(* Logix 5000 project; controller SFC_Machine_Cycle_Portfolio vendor 1 type 14 code 196 rev 36.11; software revision 36.00 *)

TASK MainTask (continuous, watchdog 500 ms) : MainProgram

MODULES
   Local : vendor 1 type 14 code 196 (5069 0, rev 36.11)
END_MODULES

VAR_GLOBAL   (* controller tags *)
   Cycle_Active : BOOL;
   Cycle_Start_Request : BOOL;
   Fault_Active : BOOL;
   Machine_Ready : BOOL;
   Mode_Auto : BOOL;
   PB_Reset : BOOL;
   PB_Start : BOOL;
   PB_Stop : BOOL;
   Stop_Request : BOOL;
END_VAR

PROGRAM MainProgram   (* main routine MainRoutine *)
VAR
   A_Unclamp : SFC_ACTION := (Status := 16#0020_0000, PauseTimer := 1);
   Action_000 : SFC_ACTION := (Status := 16#0020_0000, PauseTimer := 1);
   Clamp_Cmd : BOOL;
   Clamp_Extended_LS : BOOL;
   Clamp_Retracted_LS : BOOL;
   Clamp_Timeout_Fault : BOOL;
   Drill_At_Depth_LS : BOOL;
   Drill_At_Home_LS : BOOL;
   Drill_Fwd_Cmd : BOOL;
   Drill_Retract : SFC_STEP := (Status := 16#0020_0000, PauseTimer := 1);
   Drill_Rev_Cmd : BOOL;
   DrillFwd_Timeout_Fault : BOOL;
   DrillRev_Timeout_Fault : BOOL;
   Eject_Cmd : BOOL;
   Eject_Extend : SFC_STEP := (Status := 16#0020_0000, PauseTimer := 1);
   Eject_Extended_LS : BOOL;
   Eject_Retracted_LS : BOOL;
   EjectExtend_Timeout_Fault : BOOL;
   EjectRetract_Timeout_Fault : BOOL;
   Machine_State : DINT;   // 0 = idle 10 = Clamp 20 = Drill Foward 30 = Drill Retract 40 = Unclamp 50 = Eject Extended 60 = Eject Retract 70 = Complete
   Sim_Enable : BOOL;
   Step_Clamp_Active : BOOL;
   Step_Complete_Active : BOOL;
   Step_DrillFwd_Active : BOOL;
   Step_DrillRev_Active : BOOL;
   Step_EjectExtend_Active : BOOL;
   Step_EjectRetract_Active : BOOL;
   Step_Idle_Active : BOOL;
   Step_Unclamp_Active : BOOL;
   T_Clamp_Extend : TIMER := (PRE := 1000);
   T_Clamp_Retract : TIMER := (PRE := 1000);
   T_Clamp_Timeout : TIMER := (PRE := 3000);
   T_Drill_Fwd : TIMER := (PRE := 3000);
   T_Drill_Rev : TIMER := (PRE := 1500);
   T_DrillFwd_Timeout : TIMER := (PRE := 4000);
   T_DrillRev_Timeout : TIMER := (PRE := 4000);
   T_Eject_Extend : TIMER := (PRE := 1000);
   T_Eject_Retract : TIMER := (PRE := 1000);
   T_EjectExtend_Timeout : TIMER := (PRE := 3000);
   T_EjectRetract_Timeout : TIMER := (PRE := 3000);
   Tran_000 : BOOL;
   Tran_001 : BOOL;
   Unclamp : SFC_STEP := (Status := 16#0020_0000, PauseTimer := 1);
END_VAR

ROUTINE Faults   (* ladder *)
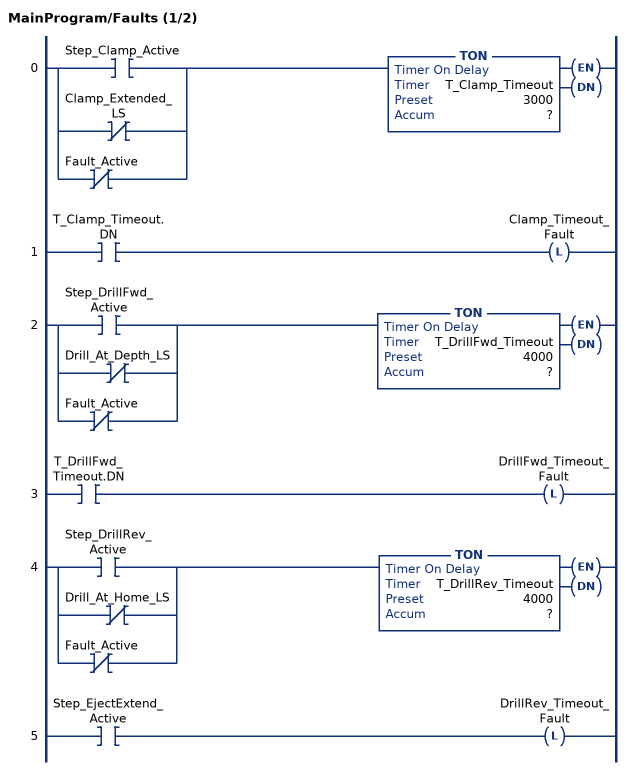
   0: [XIC(Step_Clamp_Active) ,XIO(Clamp_Extended_LS) ,XIO(Fault_Active) ]TON(T_Clamp_Timeout,?,?);
   1: XIC(T_Clamp_Timeout.DN)OTL(Clamp_Timeout_Fault);
   2: [XIC(Step_DrillFwd_Active) ,XIO(Drill_At_Depth_LS) ,XIO(Fault_Active) ]TON(T_DrillFwd_Timeout,?,?);
   3: XIC(T_DrillFwd_Timeout.DN)OTL(DrillFwd_Timeout_Fault);
   4: [XIC(Step_DrillRev_Active) ,XIO(Drill_At_Home_LS) ,XIO(Fault_Active) ]TON(T_DrillRev_Timeout,?,?);
   5: XIC(Step_EjectExtend_Active)OTL(DrillRev_Timeout_Fault);
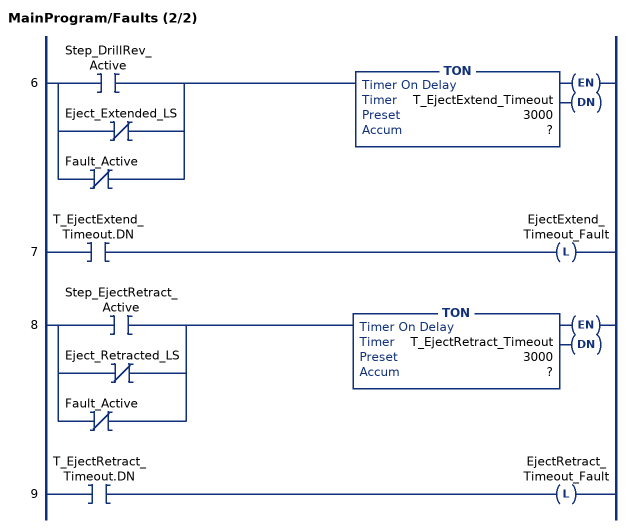
   6: [XIC(Step_DrillRev_Active) ,XIO(Eject_Extended_LS) ,XIO(Fault_Active) ]TON(T_EjectExtend_Timeout,?,?);
   7: XIC(T_EjectExtend_Timeout.DN)OTL(EjectExtend_Timeout_Fault);
   8: [XIC(Step_EjectRetract_Active) ,XIO(Eject_Retracted_LS) ,XIO(Fault_Active) ]TON(T_EjectRetract_Timeout,?,?);
   9: XIC(T_EjectRetract_Timeout.DN)OTL(EjectRetract_Timeout_Fault);
END_ROUTINE

ROUTINE Machine_SFC   (* sequential function chart *)
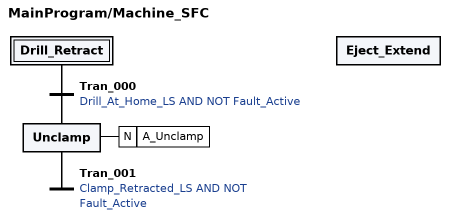
   INITIAL_STEP Drill_Retract:
   END_STEP
   TRANSITION Tran_000 FROM Drill_Retract TO Unclamp
      := Drill_At_Home_LS AND NOT Fault_Active
   END_TRANSITION
   STEP Unclamp:
      ACTION A_Unclamp (N):
         Machine_State := 40;
         Cycle_Active:= 1;
         
         Step_Idle_Active:= 0;
         Step_Clamp_Active:= 0;
         Step_DrillFwd_Active:= 0;
         Step_DrillRev_Active:= 0;
         Step_Unclamp_Active:= 1;
         Step_EjectExtend_Active:= 0;
         Step_EjectRetract_Active:= 0;
         Step_Complete_Active:= 0;
         
         Clamp_Cmd:= 0;
         Drill_Fwd_Cmd:= 0;
         Drill_Rev_Cmd:= 0;
         Eject_Cmd:= 0;
      END_ACTION
   END_STEP
   TRANSITION Tran_001 FROM Unclamp TO ()
      := Clamp_Retracted_LS AND NOT Fault_Active
   END_TRANSITION
   STEP Eject_Extend:
   END_STEP
END_ROUTINE

ROUTINE MainRoutine   (* ladder *)
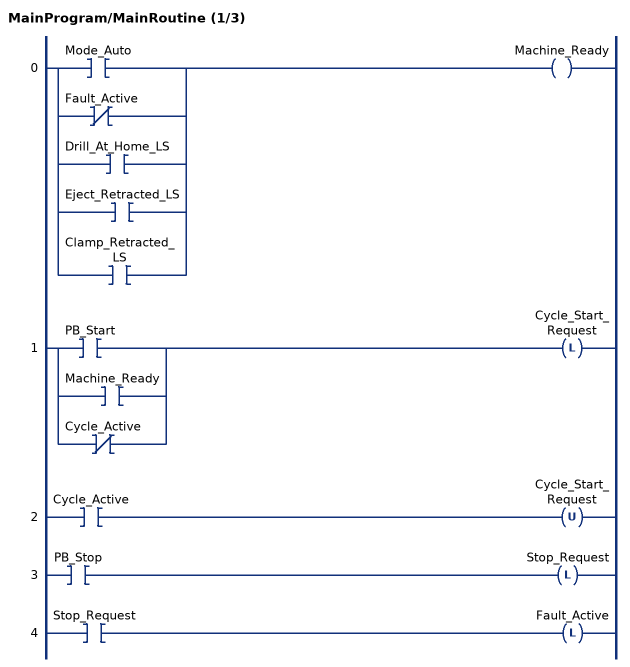
   0: [XIC(Mode_Auto) ,XIO(Fault_Active) ,XIC(Drill_At_Home_LS) ,XIC(Eject_Retracted_LS) ,XIC(Clamp_Retracted_LS) ]OTE(Machine_Ready);
   1: [XIC(PB_Start) ,XIC(Machine_Ready) ,XIO(Cycle_Active) ]OTL(Cycle_Start_Request);
   2: XIC(Cycle_Active)OTU(Cycle_Start_Request);
   3: XIC(PB_Stop)OTL(Stop_Request);
   4: XIC(Stop_Request)OTL(Fault_Active);
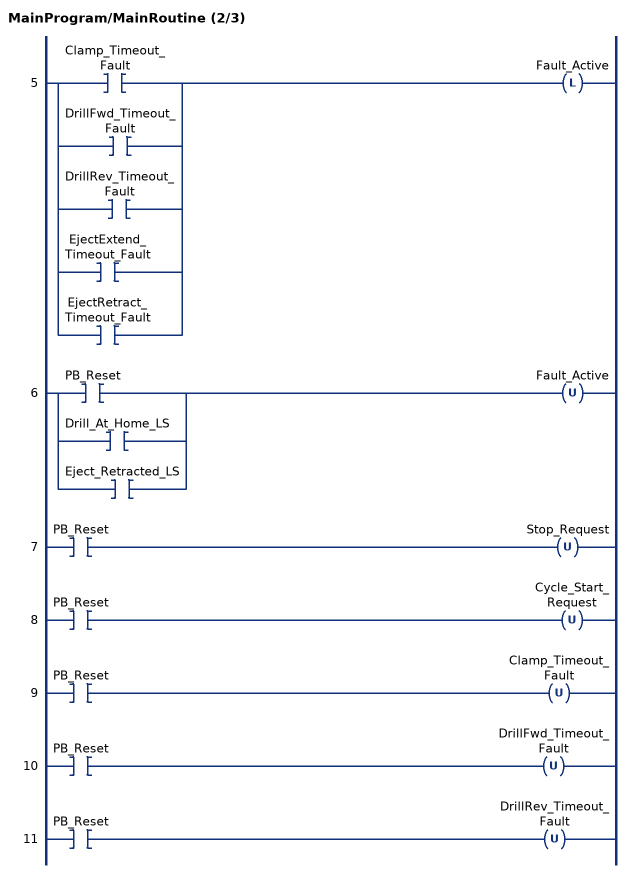
   5: [XIC(Clamp_Timeout_Fault) ,XIC(DrillFwd_Timeout_Fault) ,XIC(DrillRev_Timeout_Fault) ,XIC(EjectExtend_Timeout_Fault) ,XIC(EjectRetract_Timeout_Fault) ]OTL(Fault_Active);
   6: [XIC(PB_Reset) ,XIC(Drill_At_Home_LS) ,XIC(Eject_Retracted_LS) ]OTU(Fault_Active);
   7: XIC(PB_Reset)OTU(Stop_Request);
   8: XIC(PB_Reset)OTU(Cycle_Start_Request);
   9: XIC(PB_Reset)OTU(Clamp_Timeout_Fault);
   10: XIC(PB_Reset)OTU(DrillFwd_Timeout_Fault);
   11: XIC(PB_Reset)OTU(DrillRev_Timeout_Fault);
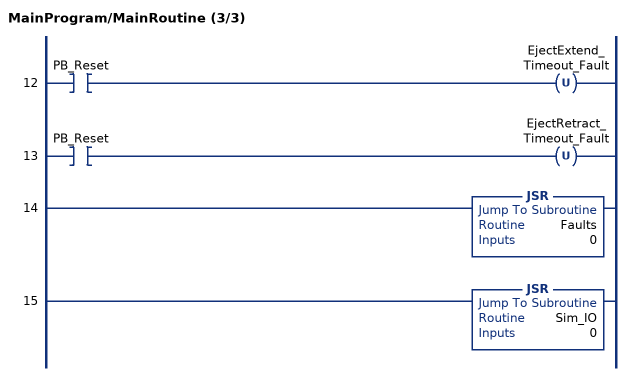
   12: XIC(PB_Reset)OTU(EjectExtend_Timeout_Fault);
   13: XIC(PB_Reset)OTU(EjectRetract_Timeout_Fault);
   14: JSR(Faults,0);
   15: JSR(Sim_IO,0);
END_ROUTINE

ROUTINE Sim_IO   (* ladder *)
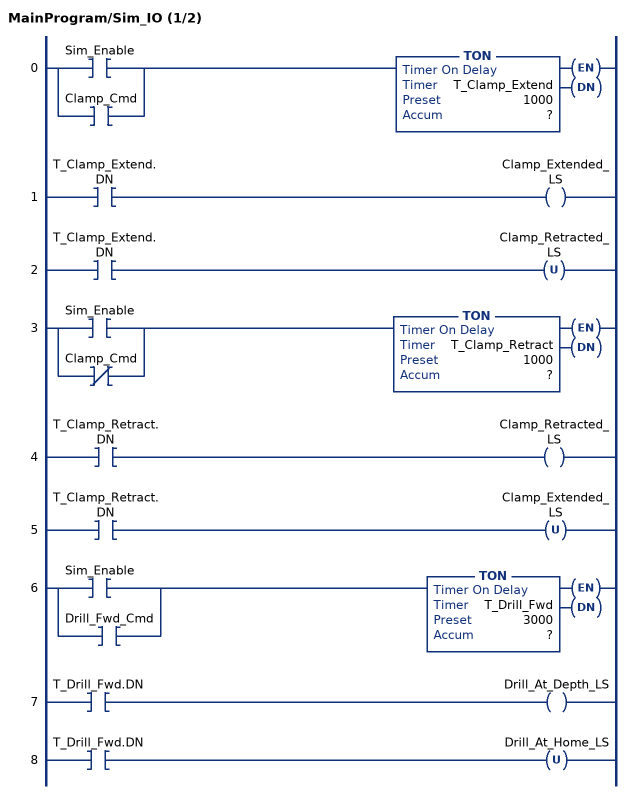
   0: [XIC(Sim_Enable) ,XIC(Clamp_Cmd) ]TON(T_Clamp_Extend,?,?);
   1: XIC(T_Clamp_Extend.DN)OTE(Clamp_Extended_LS);
   2: XIC(T_Clamp_Extend.DN)OTU(Clamp_Retracted_LS);
   3: [XIC(Sim_Enable) ,XIO(Clamp_Cmd) ]TON(T_Clamp_Retract,?,?);
   4: XIC(T_Clamp_Retract.DN)OTE(Clamp_Retracted_LS);
   5: XIC(T_Clamp_Retract.DN)OTU(Clamp_Extended_LS);
   6: [XIC(Sim_Enable) ,XIC(Drill_Fwd_Cmd) ]TON(T_Drill_Fwd,?,?);
   7: XIC(T_Drill_Fwd.DN)OTE(Drill_At_Depth_LS);
   8: XIC(T_Drill_Fwd.DN)OTU(Drill_At_Home_LS);
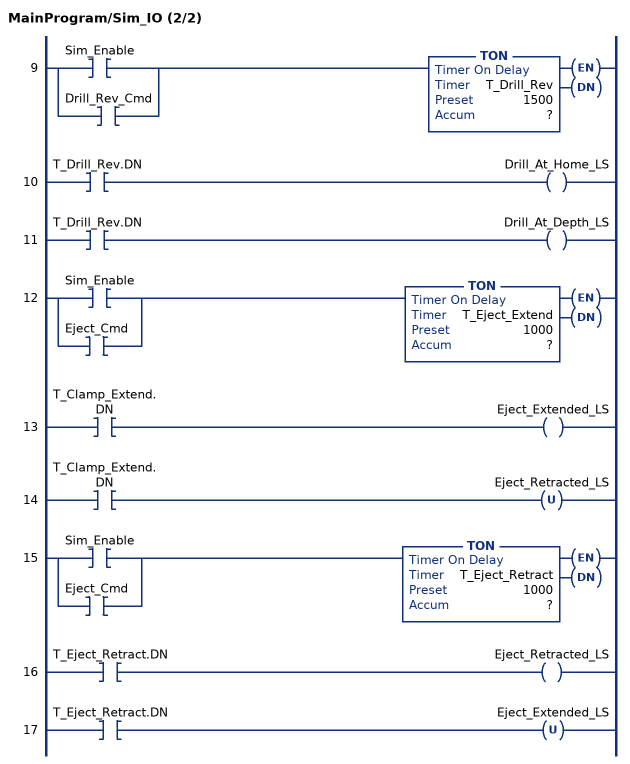
   9: [XIC(Sim_Enable) ,XIC(Drill_Rev_Cmd) ]TON(T_Drill_Rev,?,?);
   10: XIC(T_Drill_Rev.DN)OTE(Drill_At_Home_LS);
   11: XIC(T_Drill_Rev.DN)OTE(Drill_At_Depth_LS);
   12: [XIC(Sim_Enable) ,XIC(Eject_Cmd) ]TON(T_Eject_Extend,?,?);
   13: XIC(T_Clamp_Extend.DN)OTE(Eject_Extended_LS);
   14: XIC(T_Clamp_Extend.DN)OTU(Eject_Retracted_LS);
   15: [XIC(Sim_Enable) ,XIC(Eject_Cmd) ]TON(T_Eject_Retract,?,?);
   16: XIC(T_Eject_Retract.DN)OTE(Eject_Retracted_LS);
   17: XIC(T_Eject_Retract.DN)OTU(Eject_Extended_LS);
END_ROUTINE
END_PROGRAM
